FUNCTION_BLOCK FB_SetOutputBuffer
VAR_INPUT
	OutputBufferAddress				: PVOID;
	PacketAddress					: PVOID;
	SizeOfPacket					: UDINT;
END_VAR
VAR_OUTPUT
	nPacketLenght					: UDINT;
END_VAR
VAR
END_VAR

nPacketLenght := SizeOfPacket;
MEMCPY(OutputBufferAddress, 
		PacketAddress, 
		SizeOfPacket);
		
(*nPacketLenght := nPacketLenght + 1;
MEMSET(OutputBufferAddress + nPacketLenght,
	13,
	1);
	
nPacketLenght := nPacketLenght + 1;
MEMSET(OutputBufferAddress + nPacketLenght,
	10,
	1);
	*)

END_FUNCTION_BLOCK

(* stored: Version 1.1.0.1, ProductVersion 3.1.4024.2
   POU FB_SetOutputBuffer: Id {5aa13791-2dd5-4225-91b0-8b40f46058f0}, SpecialFunc None *)
